FUNCTION_BLOCK FB_GetPosition
VAR_INPUT
	bEnable		: BOOL;
END_VAR

VAR_IN_OUT
	AxisRef	 	: AXIS_REF; // Referência ao eixo do motor
END_VAR

VAR_OUTPUT
	bError		: BOOL;
	nErrorID	: UDINT;
	rPosition 	: LREAL; // Posição atual do motor
END_VAR
VAR
	ReadStatus : MC_ReadActualPosition; // Comando para leitura da posição
END_VAR

// Configura o comando para ler a posição atual do motor
ReadStatus(
	Enable 		:= bEnable,
	Axis 		:= AxisRef,
    Error  		=> bError,
    ErrorID  	=> nErrorID,
    Position 	=> rPosition
);
	
// Atualiza a variável de saída com a posição do motor
rPosition := ReadStatus.Position;

END_FUNCTION_BLOCK

(* stored: Version 1.1.0.1, ProductVersion 3.1.4024.12
   POU FB_GetPosition: Id {68a6d836-e904-4f20-8ca3-04799987088a}, SpecialFunc None *)
